Omron CX-Programmer project NewProject (CX-Programmer 9.61)

# PLC NewPLC1: CP1H XA

## Global symbols (name address type ; comment)
10.00 BOOL  ; MERAH 1
0.00 BOOL  ; START
0.01 BOOL  ; STOP
100.00 BOOL  ; SYSTEM ON
100.01 BOOL  ; SYSTEM OFF
10.01 BOOL  ; KUNING 1
10.02 BOOL  ; HIJAU 1
10.03 BOOL  ; MERAH 2
10.04 BOOL  ; KUNING 2
10.05 BOOL  ; HIJAU 2
10.06 BOOL  ; MERAH 3
10.07 BOOL  ; KUNING 3
10.08 BOOL  ; HIJAU 3
10.09 BOOL  ; MERAH 4
10.10 BOOL  ; KUNING 4
10.11 BOOL  ; HIJAU 4
60 CHANNEL  ; DATA
D0 CHANNEL  ; DATA
W0.00 BOOL  ; HIJAU 1
W0.01 BOOL  ; KUNING 1
W0.02 BOOL  ; MERAH 1

## Program NewProgram1 (cyclic task 0)

### Section Section1

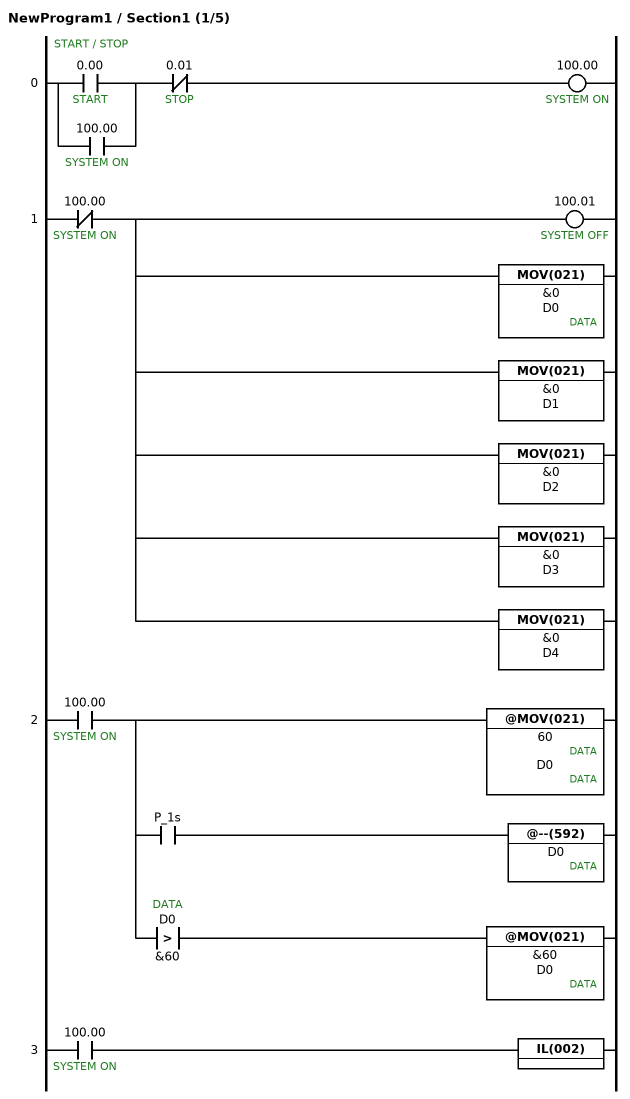
; rung 0: START / STOP
LD 0.00  ; START
OR 100.00  ; SYSTEM ON
ANDNOT 0.01  ; STOP
OUT 100.00  ; SYSTEM ON
; rung 1
LDNOT 100.00  ; SYSTEM ON
OUT 100.01  ; SYSTEM OFF
MOV(021) &0 D0  ; DATA
MOV(021) &0 D1
MOV(021) &0 D2
MOV(021) &0 D3
MOV(021) &0 D4
; rung 2
LD 100.00  ; SYSTEM ON
OUT TR0
@MOV(021) 60 D0  ; DATA
AND P_1s
@--(592) D0  ; DATA
LD TR0
AND>(320) D0 &60  ; DATA
@MOV(021) &60 D0  ; DATA
; rung 3
LD 100.00  ; SYSTEM ON
IL(002)

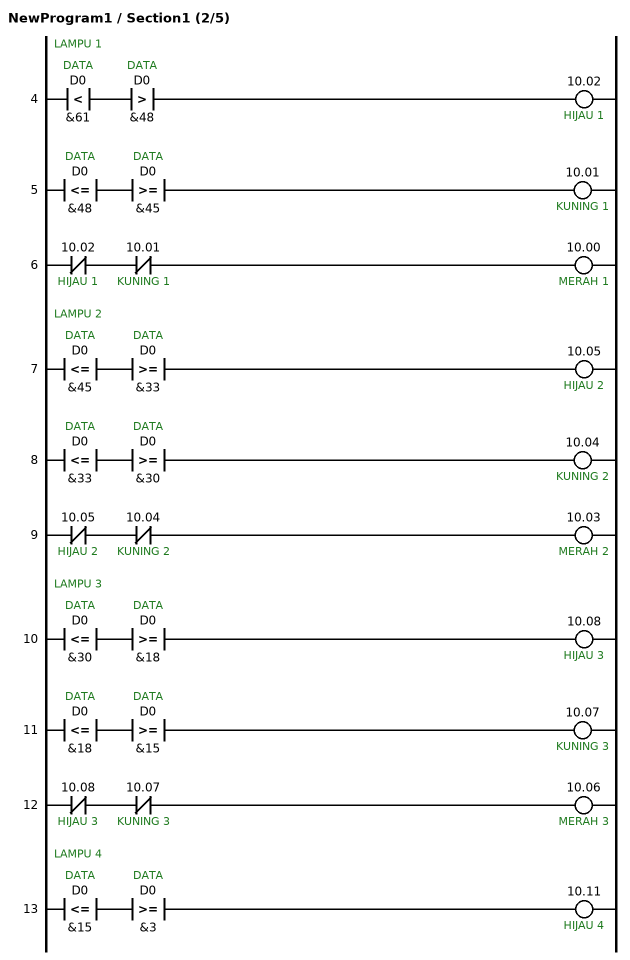
; rung 4: LAMPU 1
LD<(310) D0 &61  ; DATA
AND>(320) D0 &48  ; DATA
OUT 10.02  ; HIJAU 1
; rung 5
LD<=(315) D0 &48  ; DATA
AND>=(325) D0 &45  ; DATA
OUT 10.01  ; KUNING 1
; rung 6
LDNOT 10.02  ; HIJAU 1
ANDNOT 10.01  ; KUNING 1
OUT 10.00  ; MERAH 1
; rung 7: LAMPU 2
LD<=(315) D0 &45  ; DATA
AND>=(325) D0 &33  ; DATA
OUT 10.05  ; HIJAU 2
; rung 8
LD<=(315) D0 &33  ; DATA
AND>=(325) D0 &30  ; DATA
OUT 10.04  ; KUNING 2
; rung 9
LDNOT 10.05  ; HIJAU 2
ANDNOT 10.04  ; KUNING 2
OUT 10.03  ; MERAH 2
; rung 10: LAMPU 3
LD<=(315) D0 &30  ; DATA
AND>=(325) D0 &18  ; DATA
OUT 10.08  ; HIJAU 3
; rung 11
LD<=(315) D0 &18  ; DATA
AND>=(325) D0 &15  ; DATA
OUT 10.07  ; KUNING 3
; rung 12
LDNOT 10.08  ; HIJAU 3
ANDNOT 10.07  ; KUNING 3
OUT 10.06  ; MERAH 3
; rung 13: LAMPU 4
LD<=(315) D0 &15  ; DATA
AND>=(325) D0 &3  ; DATA
OUT 10.11  ; HIJAU 4

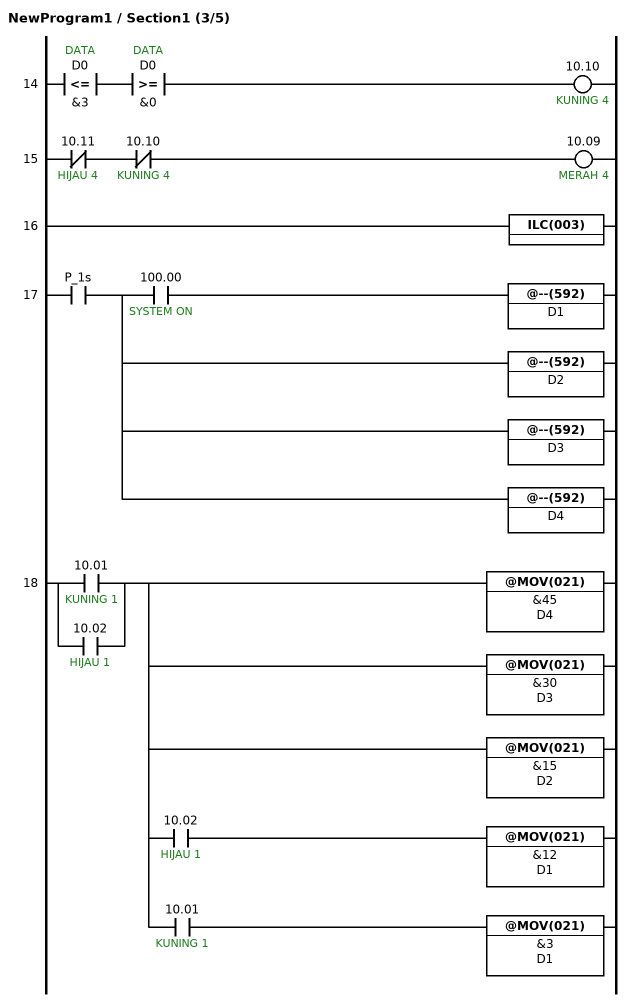
; rung 14
LD<=(315) D0 &3  ; DATA
AND>=(325) D0 &0  ; DATA
OUT 10.10  ; KUNING 4
; rung 15
LDNOT 10.11  ; HIJAU 4
ANDNOT 10.10  ; KUNING 4
OUT 10.09  ; MERAH 4
; rung 16
ILC(003)
; rung 17
LD P_1s
OUT TR0
AND 100.00  ; SYSTEM ON
@--(592) D1
LD TR0
@--(592) D2
@--(592) D3
@--(592) D4
; rung 18
LD 10.01  ; KUNING 1
OR 10.02  ; HIJAU 1
OUT TR0
@MOV(021) &45 D4
@MOV(021) &30 D3
@MOV(021) &15 D2
AND 10.02  ; HIJAU 1
@MOV(021) &12 D1
LD TR0
AND 10.01  ; KUNING 1
@MOV(021) &3 D1

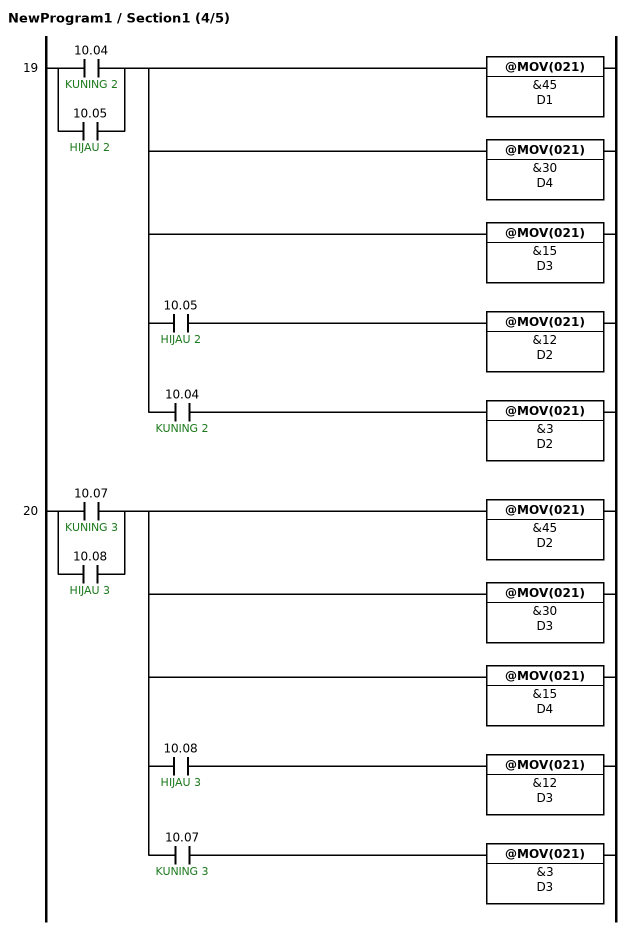
; rung 19
LD 10.04  ; KUNING 2
OR 10.05  ; HIJAU 2
OUT TR0
@MOV(021) &45 D1
@MOV(021) &30 D4
@MOV(021) &15 D3
AND 10.05  ; HIJAU 2
@MOV(021) &12 D2
LD TR0
AND 10.04  ; KUNING 2
@MOV(021) &3 D2
; rung 20
LD 10.07  ; KUNING 3
OR 10.08  ; HIJAU 3
OUT TR0
@MOV(021) &45 D2
@MOV(021) &30 D3
@MOV(021) &15 D4
AND 10.08  ; HIJAU 3
@MOV(021) &12 D3
LD TR0
AND 10.07  ; KUNING 3
@MOV(021) &3 D3

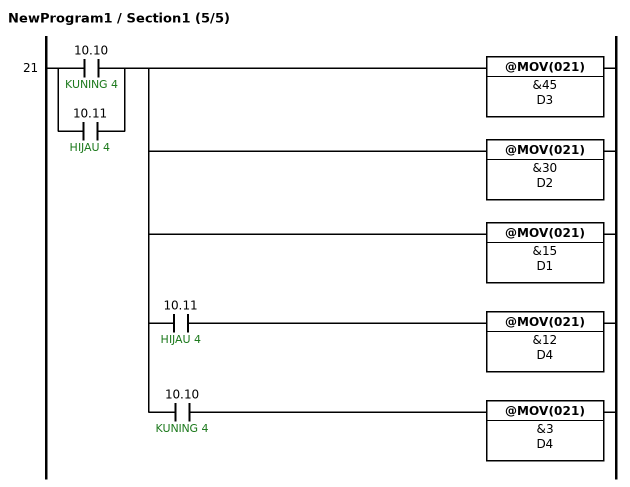
; rung 21
LD 10.10  ; KUNING 4
OR 10.11  ; HIJAU 4
OUT TR0
@MOV(021) &45 D3
@MOV(021) &30 D2
@MOV(021) &15 D1
AND 10.11  ; HIJAU 4
@MOV(021) &12 D4
LD TR0
AND 10.10  ; KUNING 4
@MOV(021) &3 D4

### Section END
; rung 0
END(001)